screen "TAKT  TIME OLD" 800x480, template "Comum"
   IOField "I/O field_1" at 506,128 size 150x39; FormatPattern 999
      ProcessValue <- "Multiplo_Uso_DB_CONTAGEM_CABINAS"
   TextField "Text field_1" at 30,109 size 222x47; Text 'PRODUÇÃO'
   TextField "Text field_2" at 38,185 size 103x47; Text 'TAKT'
   Button "Button_1" at 677,412 size 121x68; TextOff 'VOLTAR'
      on Change: ActivateScreen("PRODUCAO", 0)
   TextField "Text field_3" at 31,250 size 142x47; Text 'INICIO'
   IOField "I/O field_3" at 420,249 size 360x44; FormatPattern 99999999999999999999
      ProcessValue <- "Multiplo_Uso_DB_INICIO_JORNADA"
   IOField "I/O field_2" at 602,182 size 78x50; HelpText '1 ds'; FormatPattern 99; Unit m
      ProcessValue <- "Multiplo_Uso_DB_IHM_TAKT_MINUTOS"
   IOField "I/O field_6" at 690,182 size 78x50; HelpText '1 ds'; FormatPattern 99; Unit s
      ProcessValue <- "Multiplo_Uso_DB_IHM_TAKT_SEGUNDOS"
   TextField "Text field_6" at 677,191 size 14x32; Text ':'
   TextField "Text field_9" at 297,12 size 212x47; Text 'TAKT TIME'
   IOField "I/O field_8" at 390,420 size 78x50; HelpText '1 ds'; FormatPattern 99; Unit s
      ProcessValue <- "Multiplo_Uso_DB_IHM_Tempo_Aviso2"
   TextField "Text field_7" at 10,420 size 132x47; Text 'Aviso1'
   TextField "Text field_8" at 250,420 size 132x47; Text 'Aviso2'
   IOField "I/O field_7" at 140,420 size 100x50; HelpText '1 ds'; FormatPattern 999; Unit s
      ProcessValue <- "Multiplo_Uso_DB_IHM_Tempo_Aviso1"
   IOField "I/O field_9" at 344,128 size 150x39; FormatPattern 999
      ProcessValue <- "Multiplo_Uso_DB_TOTAL_CABINAS_TURNO"
   TextField "Text field_10" at 353,101 size 132x32; Text 'OBJETIVO'
   TextField "Text field_11" at 514,100 size 150x32; Text 'REALIZADO'
   Button "Button_2" at 687,124 size 96x42; TextOff 'ZERAR CONTAGEM'
      on Press: SetBit("Multiplo_Uso_DB_IHM_Zerar_Contagem")
      on Release: ResetBit("Multiplo_Uso_DB_IHM_Zerar_Contagem")
   Button "Button_3" at 280,190 size 96x42; TextOff 'ZERAR TAKT'
      on Press: SetBit("Multiplo_Uso_DB_IHM_Zerar_Takt")
      on Release: ResetBit("Multiplo_Uso_DB_IHM_Zerar_Takt")
   Group "Group" at 10,309 size 780x51
   Group "Group_1" at 10,367 size 780x50
   TextField "Text field_4" at 31,370 size 78x47; Text 'FIM'
   IOField "I/O field_4" at 420,313 size 360x44; FormatPattern 99999999999999999999
      ProcessValue <- "Multiplo_Uso_DB_INICIO_ALMOÇO"
   IOField "I/O field_5" at 420,371 size 360x40; FormatPattern 99999999999999999999
      ProcessValue <- "Multiplo_Uso_DB_FINAL_JORNADA"
   TextField "Text field_5" at 29,309 size 198x47; Text 'REFEIÇÃO'

screen "ANDON OLD" 800x480, template "Comum"
   TextField "Text field_1" at 312,13 size 146x47; Text 'ANDON'
   Group "Group" at 10,130 size 780x326; Picture "ESTACOES8_1"
   IOField "I/O field_1" at 190,84 size 420x160; FormatPattern 9999
      ProcessValue <- "DB_Global_Sistema_TEMPO_TAKT"
   GraphicIOField "PlotLight_Round_G" at 41,337 size 50x50; PictureOff "PilotLight_Round_G_On_256c"; PictureOn "PilotLight_Round_R_On_256c"
      ProcessValue <- "DB_Global_Sistema_Apoio_OP10"
   GraphicIOField "PlotLight_Round_G_1" at 125,337 size 50x50; PictureOff "PilotLight_Round_G_On_256c"; PictureOn "PilotLight_Round_R_On_256c"
      ProcessValue <- "DB_Global_Sistema_Apoio_OP20"
   GraphicIOField "PlotLight_Round_G_2" at 221,337 size 50x50; PictureOff "PilotLight_Round_G_On_256c"; PictureOn "PilotLight_Round_R_On_256c"
      ProcessValue <- "DB_Global_Sistema_Apoio_OP30"
   GraphicIOField "PlotLight_Round_G_3" at 316,337 size 50x50; PictureOff "PilotLight_Round_G_On_256c"; PictureOn "PilotLight_Round_R_On_256c"
      ProcessValue <- "DB_Global_Sistema_Apoio_OP40"
   GraphicIOField "PlotLight_Round_G_4" at 421,337 size 50x50; PictureOff "PilotLight_Round_G_On_256c"; PictureOn "PilotLight_Round_R_On_256c"
      ProcessValue <- "DB_Global_Sistema_Apoio_OP50"
   GraphicIOField "PlotLight_Round_G_5" at 521,337 size 50x50; PictureOff "PilotLight_Round_G_On_256c"; PictureOn "PilotLight_Round_R_On_256c"
      ProcessValue <- "DB_Global_Sistema_Apoio_OP60"
   GraphicIOField "PlotLight_Round_G_6" at 621,337 size 50x50; PictureOff "PilotLight_Round_G_On_256c"; PictureOn "PilotLight_Round_R_On_256c"
      ProcessValue <- "DB_Global_Sistema_Apoio_OP70"
   GraphicIOField "PlotLight_Round_G_7" at 715,337 size 50x50; PictureOff "PilotLight_Round_G_On_256c"; PictureOn "PilotLight_Round_R_On_256c"
      ProcessValue <- "DB_Global_Sistema_Apoio_OP80"
   Button "Button_1" at 677,412 size 121x68; TextOff 'VOLTAR'
      on Change: ActivateScreen("PRODUCAO", 0)
   GraphicView "Graphic view_2" at 711,275 size 50x45; Picture "PilotLight_Square_R_On_256c"
      Appearance <- "23U05_Cabine_Retirada"
      Visibility <- "23U05_Cabine_Retirada"
   GraphicView "Graphic view_1" at 10,130 size 780x326; Picture "ESTACOES8_1"
   TextField "Text field_2" at 49,289 size 47x20; Text 'OP.10'
   TextField "Text field_3" at 130,289 size 47x20; Text 'OP.20'
   TextField "Text field_4" at 226,289 size 47x20; Text 'OP.30'
   TextField "Text field_5" at 322,289 size 47x20; Text 'OP.40'
   TextField "Text field_6" at 421,289 size 47x20; Text 'OP.50'
   TextField "Text field_7" at 524,289 size 47x20; Text 'OP.60'
   TextField "Text field_8" at 624,289 size 47x20; Text 'OP.70'
   TextField "Text field_9" at 715,289 size 47x20; Text 'OP.80'

screen "ALARMES" 800x480, template "Comum"
   TextField "Text field_1" at 311,16 size 186x47; Text 'ALARMES'
   AlarmView "Alarm view_1" at 1,78 size 796x358
   IOField "I/O field_1" at 698,437 size 96x40; FormatPattern 999
      ProcessValue <- "ALARMES_DB_DBW0"
   Button "Button_6" at 7,438 size 164x37; TextOff 'MAIN'
      on Change: ActivateScreen("Main", 0)

screen "Ajustes do Sistema OLD" 800x480, template "Comum"
   TextField "Text field_9" at 297,12 size 184x47; Text 'AJUSTES'
   TextField "Text field_1" at 40,130 size 263x25; Text 'VELOCIDADE DE PROCESSO'
   TextField "Text field_2" at 40,163 size 170x25; Text 'VELOCIDADE JOG'
   TextField "Text field_3" at 40,194 size 208x25; Text 'AVANÇO POR CABINA'
   IOField "I/O field_1" at 290,130 size 96x32; FormatPattern 99; Unit mm/s
      ProcessValue <- "Multiplo_Uso_DB_IHM_Velocidade_Automatico"
   IOField "I/O field_2" at 290,160 size 96x32; FormatPattern 99; Unit mm/s
      ProcessValue <- "Multiplo_Uso_DB_IHM_Velocidade_Manual"
   IOField "I/O field_3" at 290,190 size 96x32; FormatPattern 9999; Unit mm
      ProcessValue <- "Multiplo_Uso_DB_IHM_Descolamento_Cabinas_mm"
   Button "FB_Plus_Rectangular" at 670,210 size 80x50; TextOff 'Text'; PictureOff "FB_Plus_Rectangular_Released_256c"; PictureOn "FB_Plus_Rectangular_Pressed_256c"
      on Press: SetBit("Multiplo_Uso_DB_IHM_Jog_CW")
      on Release: ResetBit("Multiplo_Uso_DB_IHM_Jog_CW")
   Button "Button_2" at 677,412 size 121x68; TextOff 'VOLTAR'
      on Press: ActivateScreen("MANUTENCAO", 0)
   Button "SB_ExitRuntime_85x64" at 130,410 size 85x64; TextOff 'Text'; PictureOff "SB_ExitRuntime_85x64_256c"
      on Click: StopRuntime(0)
   TextField "Text field_4" at 10,410 size 134x64; Text 'SAIR DO SISTEMA'
   Button "FB_Minus_Rectangular" at 550,210 size 80x50; TextOff 'Text'; PictureOff "FB_Minus_Rectangular_Released_256c"; PictureOn "FB_Minus_Rectangular_Pressed_256c"
      on Press: SetBit("Multiplo_Uso_DB_IHM_Jog_CCW")
      on Release: ResetBit("Multiplo_Uso_DB_IHM_Jog_CCW")
   Switch "Toggle_Horizontal_GN" at 610,90 size 80x50; TextOn 'MANUAL / 1'; CaptionText 'Switch'; TextOff 'AUTO / 0'; PictureOff "Toggle_Horizontal_GN_Off_256c"; PictureOn "Toggle_Horizontal_GN_On_256c"
      ProcessValue <- "Multiplo_Uso_DB_IHM_Modo_Manual"
   Switch "Toggle_Horizontal_GN_1" at 600,150 size 100x50; TextOn 'DRIVER ON / 1'; TextOff 'DRIVER OFF / 0'; CaptionText 'Switch'; PictureOff "Toggle_Horizontal_GN_Off_256c"; PictureOn "Toggle_Horizontal_GN_On_256c"
      ProcessValue <- "Multiplo_Uso_DB_IHM_HABILITA_DRIVER"
   Button "Button_1" at 297,303 size 96x42; TextOff 'ZERAR POSIÇÃO'
      on Press: SetBit("Multiplo_Uso_DB_IHM_Zerar_Posicao_Esteira")
      on Release: ResetBit("Multiplo_Uso_DB_IHM_Zerar_Posicao_Esteira")
   TextField "Text field_5" at 40,310 size 245x25; Text 'ZERAR POSIÇÃO ESTEIRA'
   TextField "Text field_6" at 38,224 size 245x25; Text 'POSIÇÃO ATUAL ESTEIRA'
   IOField "I/O field_4" at 290,222 size 96x32; FormatPattern 99999; Unit mm
      ProcessValue <- "Multiplo_Uso_DB_IHM_Posicao_Atual"

screen "ANDON" 800x480, template "Comum"
   TextField "Text field_1" at 312,13 size 146x47; Text 'ANDON'
   GraphicView "Graphic view_1" at 12,197 size 767x92; Picture "LINHA01"
   GraphicView "Graphic view_3" at 53,266 size 37x21; Picture "Right_Arrow"
   IOField "I/O field_1" at 190,359 size 165x49; FormatPattern 9999
      ProcessValue <- "DB_Global_Sistema_TEMPO_TAKT"
   TextField "Text field_12" at 13,367 size 173x34; Text 'TEMPO TAKT'
   GraphicView "Graphic view_4" at 133,266 size 37x21; Picture "Right_Arrow"
   GraphicView "Graphic view_5" at 229,266 size 37x21; Picture "Right_Arrow"
   GraphicView "Graphic view_6" at 322,266 size 37x21; Picture "Right_Arrow"
   GraphicView "Graphic view_7" at 421,266 size 37x21; Picture "Right_Arrow"
   GraphicView "Graphic view_8" at 524,266 size 37x21; Picture "Right_Arrow"
   GraphicView "Graphic view_9" at 618,266 size 37x21; Picture "Right_Arrow"
   GraphicView "Graphic view_11" at 707,266 size 37x21; Picture "Right_Arrow"
   TextField "Text field_3" at 47,233 size 47x20; Text 'OP.10'
   TextField "Text field_4" at 128,233 size 47x20; Text 'OP.20'
   TextField "Text field_5" at 224,233 size 47x20; Text 'OP.30'
   TextField "Text field_6" at 320,233 size 47x20; Text 'OP.40'
   TextField "Text field_7" at 416,233 size 47x20; Text 'OP.50'
   TextField "Text field_8" at 520,233 size 47x20; Text 'OP.60'
   TextField "Text field_9" at 615,233 size 47x20; Text 'OP.70'
   GraphicView "Graphic view_14" at 252,96 size 87x91; Picture "emergencia_1"
   GraphicView "Graphic view_2" at 697,224 size 58x37; Picture "PilotLight_Square_R_On_256c"
      Appearance <- "23U05_Cabine_Retirada"
      Visibility <- "23U05_Cabine_Retirada"
   TextField "Text field_10" at 703,233 size 47x20; Text 'OP.80'
   GraphicIOField "PlotLight_Round_G" at 46,297 size 50x50; PictureOff "PilotLight_Round_G_On_256c"; PictureOn "PilotLight_Round_R_On_256c"
      ProcessValue <- "DB_Global_Sistema_Apoio_OP10"
   GraphicIOField "PlotLight_Round_G_1" at 128,297 size 50x50; PictureOff "PilotLight_Round_G_On_256c"; PictureOn "PilotLight_Round_R_On_256c"
      ProcessValue <- "DB_Global_Sistema_Apoio_OP20"
   GraphicIOField "PlotLight_Round_G_2" at 223,297 size 50x50; PictureOff "PilotLight_Round_G_On_256c"; PictureOn "PilotLight_Round_R_On_256c"
      ProcessValue <- "DB_Global_Sistema_Apoio_OP30"
   GraphicIOField "PlotLight_Round_G_3" at 317,297 size 50x50; PictureOff "PilotLight_Round_G_On_256c"; PictureOn "PilotLight_Round_R_On_256c"
      ProcessValue <- "DB_Global_Sistema_Apoio_OP40"
   GraphicIOField "PlotLight_Round_G_4" at 415,297 size 50x50; PictureOff "PilotLight_Round_G_On_256c"; PictureOn "PilotLight_Round_R_On_256c"
      ProcessValue <- "DB_Global_Sistema_Apoio_OP50"
   GraphicIOField "PlotLight_Round_G_5" at 519,297 size 50x50; PictureOff "PilotLight_Round_G_On_256c"; PictureOn "PilotLight_Round_R_On_256c"
      ProcessValue <- "DB_Global_Sistema_Apoio_OP60"
   GraphicIOField "PlotLight_Round_G_6" at 612,297 size 50x50; PictureOff "PilotLight_Round_G_On_256c"; PictureOn "PilotLight_Round_R_On_256c"
      ProcessValue <- "DB_Global_Sistema_Apoio_OP70"
   GraphicIOField "PlotLight_Round_G_7" at 702,297 size 50x50; PictureOff "PilotLight_Round_G_On_256c"; PictureOn "PilotLight_Round_R_On_256c"
      ProcessValue <- "DB_Global_Sistema_Apoio_OP80"
   Button "Button_2" at 5,435 size 164x37; TextOff 'VOLTAR'; Authorization "Monitor"
      on Change: ActivateScreen("PRODUCAO", 0)
   GraphicView "Graphic view_10" at 68,96 size 87x91; Picture "emergencia_1"

screen "EMERGENCIA" 800x480, template "Comum"
   TextField "Text field_9" at 271,12 size 260x47; Text 'EMERGÊNCIA'
   GraphicView "Graphic view_1" at 12,197 size 767x92; Picture "LINHA01"
   GraphicView "Graphic view_6" at 53,266 size 37x21; Picture "Right_Arrow"
   GraphicView "Graphic view_7" at 133,266 size 37x21; Picture "Right_Arrow"
   GraphicView "Graphic view_8" at 229,266 size 37x21; Picture "Right_Arrow"
   GraphicView "Graphic view_9" at 322,266 size 37x21; Picture "Right_Arrow"
   GraphicView "Graphic view_11" at 421,266 size 37x21; Picture "Right_Arrow"
   GraphicView "Graphic view_12" at 524,266 size 37x21; Picture "Right_Arrow"
   GraphicView "Graphic view_13" at 618,266 size 37x21; Picture "Right_Arrow"
   GraphicView "Graphic view_14" at 707,266 size 37x21; Picture "Right_Arrow"
   TextField "Text field_3" at 47,233 size 47x20; Text 'OP.10'
   TextField "Text field_4" at 128,233 size 47x20; Text 'OP.20'
   TextField "Text field_5" at 224,233 size 47x20; Text 'OP.30'
   TextField "Text field_6" at 320,233 size 47x20; Text 'OP.40'
   TextField "Text field_7" at 416,233 size 47x20; Text 'OP.50'
   TextField "Text field_8" at 520,233 size 47x20; Text 'OP.60'
   TextField "Text field_1" at 615,233 size 47x20; Text 'OP.70'
   GraphicView "Graphic view_15" at 68,96 size 87x91; Picture "emergencia_1"
   GraphicView "Graphic view_16" at 252,96 size 87x91; Picture "emergencia_1"
   GraphicView "Graphic view_17" at 697,224 size 58x37; Picture "PilotLight_Square_R_On_256c"
      Appearance <- "23U05_Cabine_Retirada"
      Visibility <- "23U05_Cabine_Retirada"
   TextField "Text field_10" at 703,233 size 47x20; Text 'OP.80'
   GraphicView "Graphic view_2" at 47,303 size 46x38; Picture "emergencia"
      Appearance <- "Multiplo_Uso_DB_Emergencia_OP10_OK"
   GraphicView "Graphic view_3" at 129,303 size 46x38; Picture "emergencia"
      Appearance <- "Multiplo_Uso_DB_Emergencia_OP20_OK"
   GraphicView "Graphic view_4" at 224,303 size 46x38; Picture "emergencia"
      Appearance <- "Multiplo_Uso_DB_Emergencia_OP30_OK"
   GraphicView "Graphic view_5" at 319,303 size 46x38; Picture "emergencia"
      Appearance <- "Multiplo_Uso_DB_Emergencia_OP40_OK"
   TextField "Text field_12" at 13,366 size 262x34; Text 'PAINEL PRINCIPAL'
   GraphicView "Graphic view_10" at 268,364 size 50x40; Picture "emergencia"
      Appearance <- "Multiplo_Uso_DB_Emergencia_Principal_OK"
   Button "Button_2" at 6,437 size 164x37; TextOff 'VOLTAR'; Authorization "Operate"
      on Change: ActivateScreen("MANUTENCAO", 0)
   Button "Button_4" at 628,437 size 164x37; TextOff 'ALARMES'; TextOn 'STATUS CLP'
      on Release: ActivateScreen("ALARMES", 0)

screen "TAKT TIME" 800x480, template "Comum"
   TextField "Text field_9" at 297,12 size 212x47; Text 'TAKT TIME'
   Button "Button_1" at 17,435 size 164x37; TextOff 'VOLTAR'; Authorization "Monitor"
      on Change: ActivateScreen("PRODUCAO", 0)
   Group "Group" at 16,83 size 768x78
   TextField "Text field_2" at 33,110 size 187x40; Text 'PRODUÇÃO'
   IOField "I/O field_1" at 397,106 size 124x42; FormatPattern 999
      ProcessValue <- "Multiplo_Uso_DB_CONTAGEM_CABINAS"
   IOField "I/O field_9" at 253,106 size 124x42; FormatPattern 999
      ProcessValue <- "Multiplo_Uso_DB_TOTAL_CABINAS_TURNO"
   Button "Button_2" at 604,90 size 164x55; TextOff 'ZERAR CONTAGEM'
      on Press: SetBit("Multiplo_Uso_DB_IHM_Zerar_Contagem")
      on Release: ResetBit("Multiplo_Uso_DB_IHM_Zerar_Contagem")
   TextField "Text field_3" at 268,84 size 95x23; Text 'OBJETIVO'
   TextField "Text field_4" at 404,85 size 110x23; Text 'REALIZADO'
   Group "Group_1" at 17,165 size 766x62
   TextField "Text field_5" at 30,173 size 87x40; Text 'TAKT'
   TextField "Text field_6" at 451,173 size 181x40; Text 'T. Retirada'
   IOField "I/O field_2" at 116,172 size 124x42; HelpText '1 ds'; FormatPattern 99; Unit m
      ProcessValue <- "Multiplo_Uso_DB_IHM_TAKT_MINUTOS"
   IOField "I/O field_6" at 253,172 size 124x42; HelpText '1 ds'; FormatPattern 99; Unit s
      ProcessValue <- "Multiplo_Uso_DB_IHM_TAKT_SEGUNDOS"
   TextField "Text field_7" at 239,177 size 14x32; Text ':'
   IOField "I/O field_11" at 645,172 size 124x42; HelpText '1 ds'; FormatPattern 99; Unit s
      ProcessValue <- "Multiplo_Uso_DB_IHM_Tempo_Retirada"
   Group "Group_2" at 17,232 size 766x62
   Group "Group_3" at 17,299 size 766x62
   Group "Group_4" at 17,366 size 766x62
   TextField "Text field_8" at 30,239 size 122x40; Text 'INÍCIO'
   TextField "Text field_10" at 30,306 size 167x40; Text 'REFEIÇÃO'
   TextField "Text field_11" at 30,374 size 67x40; Text 'FIM'
   IOField "I/O field_3" at 432,238 size 337x44; FormatPattern 99999999999999999999
      ProcessValue <- "Multiplo_Uso_DB_INICIO_JORNADA"
   IOField "I/O field_4" at 432,305 size 337x44; FormatPattern 99999999999999999999
      ProcessValue <- "Multiplo_Uso_DB_INICIO_ALMOÇO"
   IOField "I/O field_5" at 432,371 size 337x44; FormatPattern 99999999999999999999
      ProcessValue <- "Multiplo_Uso_DB_FINAL_JORNADA"
   IOField "I/O field_8" at 461,434 size 100x38; HelpText '1 ds'; FormatPattern 99; Unit s
      ProcessValue <- "Multiplo_Uso_DB_IHM_Tempo_Aviso2"
   IOField "I/O field_7" at 266,434 size 100x38; HelpText '1 ds'; FormatPattern 999; Unit s
      ProcessValue <- "Multiplo_Uso_DB_IHM_Tempo_Aviso1"
   TextField "Text field_12" at 403,434 size 62x23; Text 'AVISO'
   TextField "Text field_15" at 417,450 size 27x23; Text '02'
   TextField "Text field_16" at 207,434 size 62x23; Text 'AVISO'
   TextField "Text field_17" at 225,450 size 27x23; Text '01'

screen "APRESENTAÇÃO" 800x480, template "Comum"
   Button "Button_1" at 9,436 size 164x37; TextOff 'MAIN'; Authorization "Monitor"
      on Release: ActivateScreen("Main", 0)
   TextField "Text field_1" at 250,10 size 311x47; Text 'APRESENTAÇÃO'
   GraphicView "Graphic view_1" at 11,105 size 768x230; Picture "logo_1"
   TextField "Text field_2" at 113,336 size 564x58; Text 'www.assistecnc.com.br'
*)